PROGRAM MAIN
VAR
END_VAR

SortYourNumbers();
SevenSegmentDisplay();

END_PROGRAM

(* stored: Version 1.1.0.1, ProductVersion 3.1.4024.12
   POU MAIN: Id {b0a9c719-782e-4845-845d-fbbd91c94122}, SpecialFunc None *)
